FUNCTION_BLOCK PUBLIC CapInsertStation
VAR_INPUT
END_VAR
VAR_OUTPUT
END_VAR
VAR
	xTrigger :BOOL := FALSE; // triggers processing
	State : eCapInsertStaState := eCapInsertStaState.eUnknown;
	NextState : eCapInsertStaState := eCapInsertStaState.eUnknown;
	ErrorReturnState :  eCapInsertStaState := eCapInsertStaState.eUnknown;
	bFirst : BOOL := TRUE;
	VUT : BYTE; //VehicleID Under Station
	DwellTimer : TON;		
	StateTimer : TON;
	PartPresentTimer : TON;
	CapInstallRetries : BYTE :=0;
	CapPickUpRetries : BYTE := 0;
	CapTorqueTime : TIME := T#250MS;
END_VAR

/// Cap station can be either Disabled or Enabled
// If Disabled, then we need to be in a state such that it is disabled but will not cause any obstacles. 
// Either in Disabled - Ready or Enabled- Ready, provide a way to account for Station enable change

IF (GVL_IO.MachineEStopped) THEN 
	State := eCapInsertStaState.eUnknown;
	NextState := eCapInsertStaState.eUnknown;	
END_IF

CASE State OF

eCapInsertStaState.eUnknown:
	   IF (GVL_IO.MC_XStartPB AND GVL_IO.MC_XAirPressureOK AND GVL_IO.MC_NotEStopped) THEN // wait for start button when powered up or PLC program restarted
		 ResetDwellTimer();	
         NextState := eCapInsertStaState.eHoming;	              
	   END_IF
	ACT_RetractSlide();
	ACT_RetractPalletHoldDown();
	Status.CapStatusMsg:= 'CapSta Unknown,Check Air/E-STOP THEN Hit Start';

eCapInsertStaState.eHoming:
    Status.StationStauts[MM_CONST.CAP_STA_HMI_STATE] := OverallStationStatus.eHoming;
	Status.CapStatusMsg:= 'Cap Station Homing';
	
	ACT_RetractSlide();
	ACT_RetractPalletHoldDown();
	DwellTimer(IN:=TRUE, PT:= T#10S);	
	IF (IsPalletHoldDownRetracted() AND IsSlideRetracted()) THEN
		ResetDwellTimer();	
		IF (NOT LotsData.Lot.CapInsertEnabled) THEN
			NextState :=  eCapInsertStaState.eDisabledReady;			
        ELSE 
            NextState :=  eCapInsertStaState.eWaitForVehicleTrigger;
		END_IF
	END_IF
    IF (DwellTimer.Q) THEN
		ResetDwellTimer();
		NextState := eCapInsertStaState.eError;
		ErrorReturnState := eCapInsertStaState.eHoming;		
	END_IF
	
	

eCapInsertStaState.eDisabledReady:
	ACT_RetractSlide();
	ACT_RetractPalletHoldDown();
	IF (LotsData.Lot.CapInsertEnabled) THEN 
		NextState := eCapInsertStaState.eUnknown; // force the operator to hit the start button if station is enabled.
	END_IF
	IF (xTrigger) THEN // vehicles that have been previously commanded to come here before station was disabled 
		NextState := eCapInsertStaState.eDepart;
	END_IF
	Status.StationStauts[MM_CONST.CAP_STA_HMI_STATE] := OverallStationStatus.eDisabled;
	Status.CapStatusMsg:= 'Cap Station Disabled and Clear for pallets to move';
	
	
eCapInsertStaState.eWaitForVehicleTrigger:
  
	IF (xTrigger) THEN //XTrigger is signaled when part arrives under the station
		NextState := eCapInsertStaState.ePalletHoldDownGoingDown;	
	    PartsData.Status[VUT].OverallStatus := ePartStatus.eReject; 		
		ResetDwellTimer();
	END_IF
	
	Status.StationStauts[MM_CONST.CAP_STA_HMI_STATE] := OverallStationStatus.eWaitingForParts;
	Status.CapStatusMsg:= 'Cap Station Waiting For Parts';

eCapInsertStaState.ePalletHoldDownGoingDown:
	ACT_EngagePalletHoldDown();
	IF (IsPalletHoldDownExtended()) THEN
		   NextState := eCapInsertStaState.ePalletHoldDownExtended;		 
           ResetDwellTimer();  
	   END_IF
	DwellTimer(IN:=TRUE, PT:= T#10S); // give a message out every 10 seconds
	IF (DwellTimer.Q) THEN
		ResetDwellTimer();
		NextState := eCapInsertStaState.eError;
		ErrorReturnState := eCapInsertStaState.ePalletHoldDownGoingDown;			
	END_IF
	
	Status.StationStauts[MM_CONST.CAP_STA_HMI_STATE] := OverallStationStatus.eRunning;
	Status.CapStatusMsg:= 'Cap Cycle In Progress';
	
eCapInsertStaState.ePalletHoldDownExtended:
   DwellTimer(IN:=TRUE, PT:= T#250MS);
   IF (DwellTimer.Q) THEN 
	   ResetDwellTimer();
       NextState := eCapInsertStaState.eCapSlideGoingDown;
   END_IF

eCapInsertStaState.eCapSlideGoingDown:
   ACT_ExtendSlide();
   IF (NOT IsSlideRetracted()) THEN 
	   NextState := eCapInsertStaState.eCapSlideExtended;
	   ResetDwellTimer();
   END_IF
   DwellTimer(IN:=TRUE, PT:= T#5S); // give a message out every 10 seconds
	IF (DwellTimer.Q) THEN
		ResetDwellTimer();
		Act_RetractSlide();  // Not wanting to spin the cap station if case of time out
		NextState := eCapInsertStaState.eError;
		ErrorReturnState := eCapInsertStaState.eCapSlideGoingDown;			
	END_IF

eCapInsertStaState.eCapSlideExtended:
   DwellTimer(IN:=TRUE, PT:= CapTorqueTime);
   IF (DwellTimer.Q OR IsSlideExtended()) THEN 
	   ResetDwellTimer();
	   UpdatePartData();	   
       NextState := eCapInsertStaState.eCapSlideGoingUp;
   END_IF

 eCapInsertStaState.eCapSlideGoingUp:
   ACT_RetractSlide();
   ResetDwellTimer();
   NextState := eCapInsertStaState.eCapSlideUp;
   
eCapInsertStaState.eCapSlideUp:
    IF (IsSlideRetracted()) THEN
	   ResetDwellTimer();
	   NextState := eCapInsertStaState.ePalletHoldDownGoingUp;
   END_IF
   
    DwellTimer(IN:=TRUE, PT:= T#10S); 
	IF (DwellTimer.Q) THEN
		ResetDwellTimer();
		NextState := eCapInsertStaState.eError;
		ErrorReturnState := eCapInsertStaState.eCapSlideGoingUp;			
	END_IF
   
eCapInsertStaState.ePalletHoldDownGoingUp:
	ACT_RetractPalletHoldDown();
	ResetDwellTimer();
	NextState := eCapInsertStaState.ePalletHoldDownUp;

eCapInsertStaState.ePalletHoldDownUp:
  
   IF (IsPalletHoldDownRetracted()) THEN
	   ResetDwellTimer();
	   NextState := eCapInsertStaState.eDepart;
   END_IF 
    DwellTimer(IN:=TRUE, PT:= T#10S); // give a message out every 10 seconds
	IF (DwellTimer.Q) THEN
		ResetDwellTimer();
		NextState := eCapInsertStaState.eError;
		ErrorReturnState := eCapInsertStaState.ePalletHoldDownGoingUp;			
	END_IF


eCapInsertStaState.eDepart:
	Stations.fbRoutePlanner.M_NotifyVehStaCmpl(StationIndex:= MM_CONST.CAP_STA, VehicleID := VUT);
	xTrigger := FALSE; // Now that we have sent a vehicle out, we should not work on it anymore 
    IF (Stations.fbCycleControl.StopRequested) THEN		
		NextState := eCapInsertStaState.eStopActive;
	ELSE
		NextState := eCapInsertStaState.eHoming;
	END_IF

eCapInsertStaState.eStopActive:
IF (NOT Stations.fbCycleControl.StopRequested) THEN		
		NextState := eCapInsertStaState.eHoming;
END_IF	
    Status.StationStauts[MM_CONST.CAP_STA_HMI_STATE] := OverallStationStatus.eCycleStop;	
    Status.CapStatusMsg:= 'Cap Stop Active, Press Start to Run';
	
eCapInsertStaState.eError:
	Status.StationStauts[MM_CONST.CAP_STA_HMI_STATE] := OverallStationStatus.eError;
	IF (GVL_IO.MC_XStartPB) THEN
		NextState := ErrorReturnState;
		ErrorReturnState := eCapInsertStaState.eUnknown;
	END_IF
	
END_CASE

IF (State <> NextState) THEN
	bFirst := TRUE;
	StateTimer(IN:=FALSE);
ELSE
	bFirst := FALSE;
END_IF

State := NextState;

ACTION ACT_EngagePalletHoldDown:
GVL_IO.CP_YPalletHoldDownExtend := TRUE;
GVL_IO.CP_YPalletHoldDownRetract := FALSE;
END_ACTION

ACTION ACT_ExtendSlide:
GVL_IO.CP_YCapSlideExtend := TRUE;
GVL_IO.CP_YCapSlideRetract := FALSE;
END_ACTION

ACTION ACT_RetractPalletHoldDown:
GVL_IO.CP_YPalletHoldDownExtend := FALSE;
GVL_IO.CP_YPalletHoldDownRetract := TRUE;
END_ACTION

ACTION ACT_RetractSlide:
GVL_IO.CP_YCapSlideExtend := FALSE;
GVL_IO.CP_YCapSlideRetract := TRUE;
END_ACTION

METHOD PUBLIC ClearVehicleTrigger : BOOL
VAR_INPUT
END_VAR
xTrigger := FALSE;
END_METHOD

METHOD PUBLIC IsFaulted : BOOL
VAR_INPUT
END_VAR
IF (LotsData.Lot.CapInsertEnabled) THEN 
	IsFaulted := (State = eCapInsertStaState.eUnknown OR State = eCapInsertStaState.eError);
ELSE 
	IsFaulted := FALSE;
END_IF
END_METHOD

METHOD PUBLIC IsPalletHoldDownExtended : BOOL
VAR_INPUT
END_VAR
IsPalletHoldDownExtended := (GVL_IO.CP_XPalletHoldDownExtended AND NOT GVL_IO.CP_XPalletHoldDownHome);
IF (NOT IsPalletHoldDownExtended) THEN 
	Status.CapStatusMsg := 'Cap Station: Check Pallet HoldDown Sensors'; 
END_IF
END_METHOD

METHOD PUBLIC IsPalletHoldDownRetracted : BOOL
VAR_INPUT
END_VAR
IsPalletHoldDownRetracted := (NOT GVL_IO.CP_XPalletHoldDownExtended AND GVL_IO.CP_XPalletHoldDownHome);
IF (NOT IsPalletHoldDownRetracted) THEN 
	Status.CapStatusMsg := 'Cap Station: Check Pallet HoldDown Sensors'; 
END_IF
END_METHOD

METHOD IsSlideExtended : BOOL
VAR_INPUT
END_VAR
IsSlideExtended := (GVL_IO.CP_XCapSlideExtended AND NOT GVL_IO.CP_XCapSlideRetracted);
IF (NOT IsSlideExtended) THEN 
	Status.CapStatusMsg := 'Cap Station: Check Slide Sensors'; 
END_IF
END_METHOD

METHOD PUBLIC IsSlideRetracted : BOOL
VAR_INPUT
END_VAR
//IsSlideRetracted := TRUE; //turnkey slide removed

IsSlideRetracted := (NOT GVL_IO.CP_XCapSlideExtended AND GVL_IO.CP_XCapSlideRetracted);
IF (NOT IsSlideRetracted) THEN 
	Status.CapStatusMsg := 'Cap Station: Check Slide Sensors'; 
END_IF
END_METHOD

PROPERTY PUBLIC Ready : BOOL
GET
IF (LotsData.Lot.CapInsertEnabled) THEN
 Ready := (State = eCapInsertStaState.eWaitForVehicleTrigger);
ELSE
	Ready := (State = eCapInsertStaState.eDisabledReady);	//we removed the physical cap station on 10/17 
END_IF
END_GET
END_PROPERTY

ACTION ResetDwellTimer:
DwellTimer(IN:=FALSE);
END_ACTION

METHOD PUBLIC ResetState : BOOL
VAR_INPUT
END_VAR
	State := eCapInsertStaState.eUnknown;
	NextState := eCapInsertStaState.eUnknown;
	ErrorReturnState := eCapInsertStaState.eUnknown;
END_METHOD

PROPERTY PUBLIC Trigger : BOOL
SET
xTrigger := Trigger;
END_SET
END_PROPERTY

METHOD PUBLIC UpdatePartData : BOOL
VAR_INPUT
END_VAR
IF ( NOT IsSlideExtended()) THEN
	PartsData.Status[VUT].OverallStatus := ePartStatus.eCapInserted;
	PartsData.Status[VUT].CapPass := TRUE;
	PartsData.Status[VUT].CapInsertTime := SYSTEMTIME_TO_STRING(Logging.fbCurrTime.systemTime);	
ELSE // there is no cap
	PartsData.Status[VUT].OverallStatus := ePartStatus.eReject;
	PartsData.Status[VUT].CapPass := FALSE;
	PartsData.Status[VUT].CapInsertTime := SYSTEMTIME_TO_STRING(Logging.fbCurrTime.systemTime);
END_IF
END_METHOD

PROPERTY PUBLIC VehicleUnderTest : BYTE
GET
VehicleUnderTest := VUT;
END_GET
SET
VUT := VehicleUnderTest;
END_SET
END_PROPERTY

END_FUNCTION_BLOCK

(* stored: Version 1.1.0.1, ProductVersion 3.1.4022.6
   POU CapInsertStation: Id {81c9b069-8f42-4f4e-84c1-86db7f85b7eb}, SpecialFunc None
   Action ACT_EngagePalletHoldDown: Id {95141e64-78f7-4867-bf7b-5bed44ebbacc}
   Action ACT_ExtendSlide: Id {1d578825-4866-4394-8f8f-fa56dc169ceb}
   Action ACT_RetractPalletHoldDown: Id {459630e6-80b4-4310-a27c-d15b3a660d34}
   Action ACT_RetractSlide: Id {fa2221e9-2918-483a-995a-ca1615d630ca}
   Method ClearVehicleTrigger: Id {989176d5-bf81-42c2-a0c0-8a0eacb996bc}
   Method IsFaulted: Id {f2bd33d3-6b53-4212-a61d-4ad059b85326}
   Method IsPalletHoldDownExtended: Id {73fe6c18-868c-43aa-bb67-6b2b57ebf00e}
   Method IsPalletHoldDownRetracted: Id {fa3344f9-dc29-4857-adab-21ba290392e4}
   Method IsSlideExtended: Id {74ad416d-3a39-497e-ad01-365b5f014f7f}
   Method IsSlideRetracted: Id {02fc8f15-02f2-4aec-843b-2d256722b895}
   Property Ready: Id {a05d8b61-4f3b-45b3-8057-31455b12851f}
   Get Get: Id {34333ac7-2221-4d33-a374-d65e0015b754}
   Action ResetDwellTimer: Id {6db09a20-8cd6-4a84-bd68-f0501f569845}
   Method ResetState: Id {75773aca-2a2e-44f3-9965-4b9bb1aa8777}
   Property Trigger: Id {2f10ab5f-92bd-4ae2-9f5b-d857e3c1dacd}
   Set Set: Id {2fda31bd-35dc-4d46-bd9d-a929e6e758a0}
   Method UpdatePartData: Id {ef3d3634-ab22-4402-bff7-d14f68097d26}
   Property VehicleUnderTest: Id {1253488d-acf7-452b-bf65-0fa3c66dae26}
   Get Get: Id {0c78b70f-f938-41af-a1a7-0a125494ecd7}
   Set Set: Id {c601952b-332a-4ce3-be39-06cc9be0ac8b} *)
